FUNCTION_BLOCK T_ListOfTests IMPLEMENTS I_ListOfTests
VAR
    {attribute 'analysis' := '-33'} // inhibit unused variable warning
    DynamicMemoryManager : FB_DynMem_Manager;
    Buffer               : FB_DynMem_Buffer(ipMemMan := DynamicMemoryManager);
    pTest                : POINTER TO I_UnitTest;
    _Count               : DINT;
    Capacity             : DINT;
END_VAR

METHOD AddTest
VAR_INPUT
    Test : I_UnitTest;
END_VAR
IF _Count = Capacity THEN
    Capacity := Capacity * 2;
    Buffer.Resize(nSize     := DINT_TO_UDINT(Capacity) * SIZEOF(PVOID),
                  bPreserve := TRUE,
                  bReset    := FALSE);

    pTest := Buffer.pBuffer;
END_IF

IF pTest = 0 THEN
    F_LogError(Source  := 'T_ListOfTests.AddTest()',
                Message := 'Buffer not initialised');
ELSE
    pTest[_Count] := Test;
    _Count        := _Count + 1;
END_IF
END_METHOD

METHOD Clear
VAR_INPUT
END_VAR
IF pTest = 0 THEN
    // Buffer was not allocated during Fb_init. Try again...
    Buffer.CreateBuffer(nSize  := DINT_TO_UDINT(Capacity) * SIZEOF(PVOID),
                        bReset := TRUE);
END_IF

Buffer.Clear();
_Count := 0;
END_METHOD

PROPERTY Count : DINT
GET
Count := _Count;
END_GET
END_PROPERTY

METHOD FB_exit : BOOL
VAR_INPUT
    bInCopyCode : BOOL; // if TRUE, the exit method is called for exiting an instance that is copied afterwards (online change).
END_VAR
IF NOT bInCopyCode THEN
    Buffer.DeleteBuffer();
    pTest := 0;
END_IF
END_METHOD

METHOD FB_init : BOOL
VAR_INPUT
    bInitRetains : BOOL; // if TRUE, the retain variables are initialized (warm start / cold start)
    bInCopyCode  : BOOL; // if TRUE, the instance afterwards gets moved into the copy code (online change)
    Capacity     : DINT;
END_VAR
Buffer.CreateBuffer(nSize  := DINT_TO_UDINT(Capacity) * SIZEOF(PVOID),
                    bReset := TRUE);

pTest := Buffer.pBuffer;

THIS^.Capacity := Capacity;
END_METHOD

METHOD GetTest : I_UnitTest
VAR_INPUT
    Index : DINT;
END_VAR
IF Index < _Count AND Index >= 0 THEN
    GetTest := pTest[Index];
END_IF
END_METHOD

END_FUNCTION_BLOCK

(* stored: Version 1.1.0.1, ProductVersion 3.1.4024.12
   POU T_ListOfTests: Id {1fcff8f0-b8c4-4bed-b839-fdb26fdb9776}, SpecialFunc None
   Folder Methods: Id {88ea0914-3836-4c42-892b-eaef76e9b52e}
   Folder Properties: Id {ebcc07c5-4fc8-427f-8482-a63a96860394}
   Method AddTest: Id {4faaef0c-95d4-47eb-bad8-5f502cf946ca}
   Method Clear: Id {392cea44-d6e9-4110-b6d9-4fed5b76a2ec}
   Property Count: Id {3952cc7c-1071-4603-8d76-4fe94cd90db2}
   Get Get: Id {0e88bdd7-52c9-4eea-969d-92abc8c68f8b}
   Method FB_exit: Id {b4bcf37e-def8-4b6e-bf9c-b2a96004e198}
   Method FB_init: Id {c7aec280-ba2a-4496-90e8-87d0d03568b6}
   Method GetTest: Id {da1f2a72-8905-472e-8ebd-a6a8733af20d} *)
